
// ===== library: MasterCopy "DataItemNumeric" =====

TYPE "DataItemNumeric"
   STRUCT
      "name" : String[20];
      category : UInt;
      value : Real;
      prevvalue : Real;
      decimal : Int;
      send : Bool;
   END_STRUCT;
END_TYPE

// ===== library: MasterCopy "DataItemBool" =====

TYPE "DataItemBool"
   STRUCT
      "name" : String[20];
      category : UInt;
      value : Bool;
      prevValue : Bool;
      send : Bool;
   END_STRUCT;
END_TYPE

// ===== library: MasterCopy "Copy of Program blocks in MTConnect" =====
// protected blocks, not shown: "MTCONNECT"

// folder: MTConnect

DATA_BLOCK "MTCData"   // DB1
{ S7_Optimized_Access := 'FALSE' }
VERSION : 0.1
   VAR
      "Bool" : Array[0..1] of "DataItemBool";
      Numeric : Array[0..1] of "DataItemNumeric";
      test : TCON_IP_v4;
   END_VAR
BEGIN
END_DATA_BLOCK

FUNCTION "SizeOf" : Void   // FC1, SCL
{ S7_Optimized_Access := 'FALSE' }
VERSION : 0.1
BEGIN
   #SizeOf := CountOfElements(#Arrayin);
END_FUNCTION

FUNCTION "TimeStamp" : Void   // FC2, SCL
{ S7_Optimized_Access := 'FALSE' }
VERSION : 0.1
BEGIN
   //  Form Timestamp for MTConnect
   //  By: Bryan Garness
   //  ISO8601 FORMAT SHDR 
   //  YYYY-MM-DDTHH:MM:SS.FFFFFFZ


   #Ret := RD_SYS_T(#DTLREAD);
   VAL_STRG(IN := #DTLREAD.YEAR,
            SIZE := 4,
            PREC := 0,
            FORMAT := 0,
            P := 1,
            OUT => #TempString);
   IF #DTLREAD.MONTH > 9 THEN
     #TempString := CONCAT(IN1 := #TempString, IN2 := '-');
     VAL_STRG(IN := #DTLREAD.MONTH,
              SIZE := 2,
              PREC := 0,
              FORMAT := 0,
              P := 1,
              OUT => #TempString2);
   ELSE
     #TempString := CONCAT(IN1 := #TempString, IN2 := '-0');
     VAL_STRG(IN := #DTLREAD.MONTH,
              SIZE := 1,
              PREC := 0,
              FORMAT := 0,
              P := 1,
              OUT => #TempString2);
   END_IF;

   #TempString := CONCAT(IN1 := #TempString, IN2 := #TempString2);
   #TempString2 := '';
   IF #DTLREAD.DAY > 9 THEN
     #TempString := CONCAT(IN1 := #TempString, IN2 := '-');
     VAL_STRG(IN := #DTLREAD.DAY,
              SIZE := 2,
              PREC := 0,
              FORMAT := 0,
              P := 1,
              OUT => #TempString2);
   ELSE
     #TempString := CONCAT(IN1 := #TempString, IN2 := '-0');
     VAL_STRG(IN := #DTLREAD.DAY,
              SIZE := 1,
              PREC := 0,
              FORMAT := 0,
              P := 1,
              OUT => #TempString2);
   END_IF;

   #TempString := CONCAT(IN1 := #TempString, IN2 := #TempString2);
   #TempString2 := '';
   #TempString := CONCAT(IN1 := #TempString, IN2 := 'T');
   IF #DTLREAD.HOUR > 9 THEN
     VAL_STRG(IN := #DTLREAD.HOUR,
              SIZE := 2,
              PREC := 0,
              FORMAT := 0,
              P := 1,
              OUT => #TempString2);
   ELSE
     #TempString := CONCAT(IN1 := #TempString, IN2 := '0');
     VAL_STRG(IN := #DTLREAD.HOUR,
              SIZE := 1,
              PREC := 0,
              FORMAT := 0,
              P := 1,
              OUT => #TempString2);
   END_IF;
   #TempString := CONCAT(IN1 := #TempString, IN2 := #TempString2);
   #TempString2 := '';
   #TempString := CONCAT(IN1 := #TempString, IN2 := ':');
   IF #DTLREAD.MINUTE > 9 THEN
     VAL_STRG(IN := #DTLREAD.MINUTE,
              SIZE := 2,
              PREC := 0,
              FORMAT := 0,
              P := 1,
              OUT => #TempString2);
   ELSE
     #TempString := CONCAT(IN1 := #TempString, IN2 := '0');
     VAL_STRG(IN := #DTLREAD.MINUTE,
              SIZE := 1,
              PREC := 0,
              FORMAT := 0,
              P := 1,
              OUT => #TempString2);
   END_IF;
   #TempString := CONCAT(IN1 := #TempString, IN2 := #TempString2);
   #TempString := CONCAT(IN1 := #TempString, IN2 := ':');
   IF #DTLREAD.SECOND > 9 THEN
     VAL_STRG(IN := #DTLREAD.SECOND,
              SIZE := 2,
              PREC := 0,
              FORMAT := 0,
              P := 1,
              OUT => #TempString2);
   ELSE
     #TempString := CONCAT(IN1 := #TempString, IN2 := '0');
     VAL_STRG(IN := #DTLREAD.SECOND,
              SIZE := 1,
              PREC := 0,
              FORMAT := 0,
              P := 1,
              OUT => #TempString2);
   END_IF;
   #TempString := CONCAT(IN1 := #TempString, IN2 := #TempString2);
   #TempString2 := '';

   #MathTemp := #DTLREAD.NANOSECOND / 1000;
   VAL_STRG(IN := #MathTemp,
            SIZE := 8,
            PREC := 6,
            FORMAT := 2,
            P := 1,
            OUT => #TempString2);
   #TempString2 := RIGHT(IN := #TempString2, L := 7);
   #TempString := CONCAT(IN1 := #TempString, IN2 := #TempString2);
   //#TempString := CONCAT(IN1 := #TempString, IN2 := 'Z');
   #UTCStamp := #TempString;
END_FUNCTION